{attribute 'GeneratedUsingTerminal: EL3751-0000-0020'}
{attribute addProperty BoxType "EL3751-0000-0020"}
{attribute addProperty Id "PAI_StatusAT %I*PAI_Status_Channel_AE4AC1047PAI_Samples_1AT %I*PAI_Samples_EEA517254PAI_TimestampAT %I*PAI_Timestamp_6DC4D2968WcStateAT %I*WcState_9091E0EB2InfoDataAT %I*InfoData_1088C70510"}
{attribute addProperty CRC "87589525"}
{attribute addProperty Size "31"}
TYPE EL3751_05388295 EXTENDS EtcSlaveTerminalBase_947E5A46 :
STRUCT
	{attribute addProperty Name "PAI_Status"}
	PAI_Status : PAI_Status_Channel_AE4AC104;
	{attribute addProperty Name "PAI_Samples_1"}
	PAI_Samples_1 : PAI_Samples_EEA51725;
	{attribute addProperty Name "PAI_Timestamp"}
	PAI_Timestamp : PAI_Timestamp_6DC4D296;
	{attribute addProperty Name "WcState"}
	WcState : WcState_9091E0EB;
	{attribute addProperty Name "InfoData"}
	InfoData : InfoData_1088C705;
END_STRUCT
END_TYPE

(* stored: Version 1.2.0.0, ProductVersion 3.1.4024.9
   DUT EL3751_05388295: Id {4f6bf136-24aa-471f-ad66-8de7c6dd2b40} *)
